// TIA Portal V16 export
// export: Created 2021-05-25T16:14:39.2264959Z, ExportSetting WithDefaults, DisplayName Totally Integrated Automation Portal, DisplayVersion V16, DisplayName TIA Portal Version Control Interface, DisplayVersion V16, DisplayName TIA Portal Openness, DisplayVersion V16, DisplayName STEP 7 Professional, DisplayVersion V16, DisplayName STEP 7 Safety, DisplayVersion V16, DisplayName WinCC Unified SCADA Engineering System, DisplayVersion V16
DATA_BLOCK "dbProfinetAlrm"   // DB4
{ S7_Optimized_Access := 'FALSE'; DB_Accessible_From_OPC_UA := 'FALSE' }
VERSION : 0.0
// stored: AutoNumber true, DBAccessibleFromOPCUA false, IsOnlyStoredInLoadMemory false, IsWriteProtectedInAS false
   VAR
      ProfiNet_Req : Bool := FALSE;
      ProfiNet_SzlID : DWord := 16#0000;
      ProfiNet_Index : Int := 16#0000;
      Profinet_RetVal : Int := 0;
      ProfiNet_Busy : Bool := FALSE;
      ProfiNet_En : Bool := FALSE;
   END_VAR
BEGIN
END_DATA_BLOCK
